FUNCTION_BLOCK MedianBlur (* openCV median blur filter *)
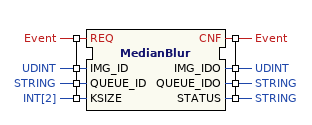
  EVENT_INPUT
    REQ WITH IMG_ID, QUEUE_ID, KSIZE;
  END_EVENT
  EVENT_OUTPUT
    CNF WITH IMG_IDO, QUEUE_IDO, STATUS;
  END_EVENT
  VAR_INPUT
    IMG_ID : UDINT;
    QUEUE_ID : STRING;
    KSIZE : ARRAY [0..1] OF INT;
  END_VAR
  VAR_OUTPUT
    IMG_IDO : UDINT;
    QUEUE_IDO : STRING;
    STATUS : STRING;
  END_VAR
END_FUNCTION_BLOCK
